(* Logix 5000 project; controller TrafficLightDemo vendor 1 type 14 code 154 rev 32.11; software revision 32.05 *)

MODULES
   Local : vendor 1 type 14 code 154 (PointIO 0, rev 32.11)
      Discrete_IO : Embedded (PointIO 1, rev 32.11, Output RPI 20 ms)
END_MODULES

VAR_GLOBAL   (* controller tags *)
   Green_Light : BOOL;
   Red_Light : BOOL;
   Step : DINT;
   T_Green : TIMER;
   T_Red : TIMER;
   T_Yellow : TIMER;
   Yellow_Light : BOOL;
END_VAR

PROGRAM Traffic_Light_Program

ROUTINE MainRoutine   (* ladder *)
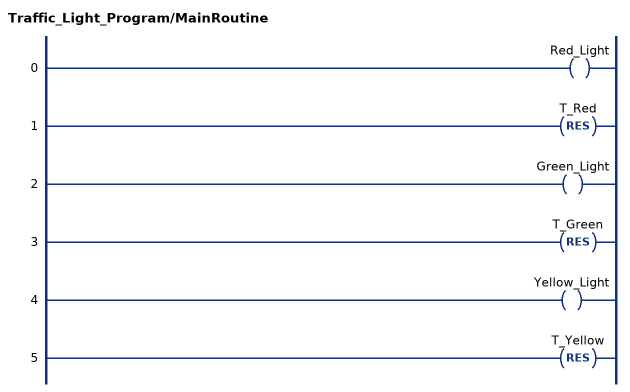
   0: OTE(Red_Light);
   1: RES(T_Red);
   2: OTE(Green_Light);
   3: RES(T_Green);
   4: OTE(Yellow_Light);
   5: RES(T_Yellow);
END_ROUTINE
END_PROGRAM
